{attribute 'GeneratedUsingTerminal: AT2026-0250-0020'}
{attribute addProperty BoxType "AT2026-0250-0020"}
{attribute addProperty Id "A_0078_AT2001_5250_0019_AT2001_5250AT2001_01D6DEDF80"}
{attribute addProperty CRC "1063729990"}
{attribute addProperty Size "80"}
TYPE A_0066_AT2026_0250_0020_AT2026_0250_3F673B46 EXTENDS AT2026_86175B41 :
STRUCT
	{attribute addProperty Name "A_0078_AT2001_5250_0019_AT2001_5250"}
	{attribute addProperty PreviousPort "A_0066(AT2026-0250-0020) (AT2026-0250) : B"}
	A_0078_AT2001_5250_0019_AT2001_5250 : AT2001_01D6DEDF;
END_STRUCT
END_TYPE

(* stored: Version 1.2.0.0, ProductVersion 3.1.4024.9
   DUT A_0066_AT2026_0250_0020_AT2026_0250_3F673B46: Id {655d7ae8-cebd-4d1d-96a1-aaecc328e420} *)
